FUNCTION_BLOCK EscreveBD
VAR_INPUT
END_VAR
VAR_OUTPUT
END_VAR
VAR
END_VAR

END_FUNCTION_BLOCK

(* stored: Version 1.1.0.1, ProductVersion 3.1.4024.13
   POU EscreveBD: Id {eae73980-1c52-4c41-a457-2040f5753823}, SpecialFunc None *)
